TYPE UDT_DevManualCtrl :
STRUCT
END_STRUCT
END_TYPE

(* stored: Version 1.1.0.1, ProductVersion 3.1.4024.4
   DUT UDT_DevManualCtrl: Id {d714b36f-2088-0809-3d4b-82ff0c73dc2f} *)
